ABB RobotStudio station: SJAKKROBOT.rspag

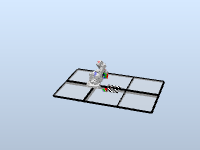
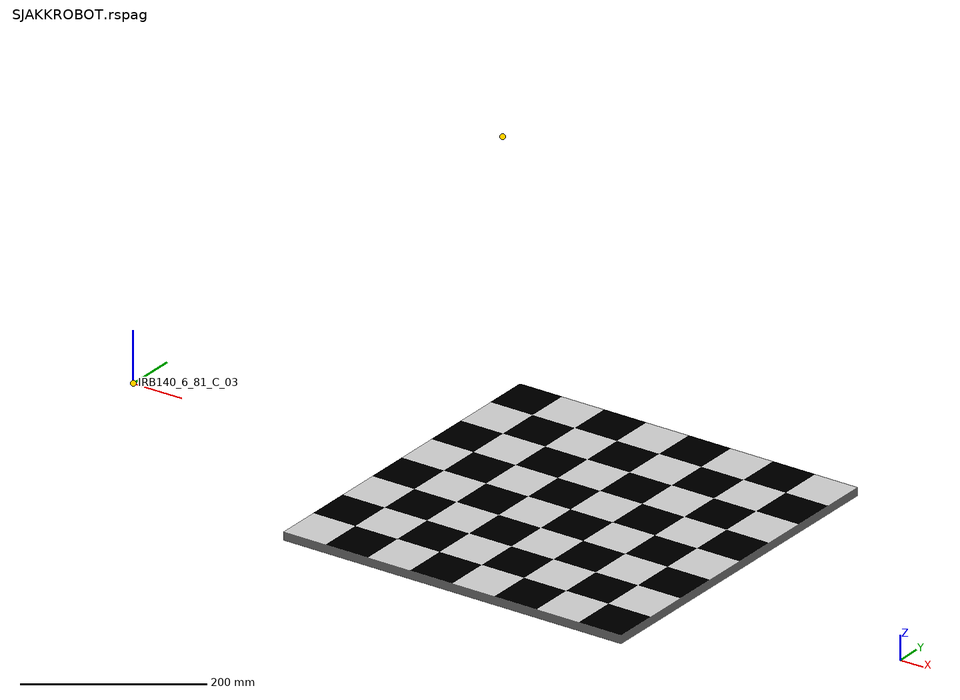
[picture v1: parts stored in the station drawn from their meshes, with robot base, taught points and paths (robot models come from the ABB library and are not in the file)]
--- station ---
Station Solution10 (saved by RobotStudio 21.2.9526.0)
Controller IRB140_6_81
  mechanical unit ROB_1: IRB140_6_81_C_03, 6 joints, base frame (0, 0, 0) mm
Layout (positions relative to the parent item):
  - IRB140_6_81_C_03 [mechanism, from Robots\IRB140_6_81_C_G_03.rslib] at (0, 0, 0) mm; joint values [1.0633, 0.4639, 0.5303, 0, 0.5766, 4.2048] (rad or m)
  - Part_1 [part], size 20 x 20 x 100 mm
  - picker [mechanism] at (210.95, 383, 290.4) mm, rotated rx -180 ry 0 rz 0 deg
      TCP picker at (0, 0, 100) mm
      links: Dummy
  - Brett [part], size 440 x 440 x 9.9 mm
  - 1 [part] at (50, 0, 0) mm, size 55 x 440 x 0 mm
  - 2 [part] at (105, 0, 0) mm, size 55 x 440 x 0 mm
  - 3 [part] at (160, 0, 0) mm, size 55 x 440 x 0 mm
  - 4 [part] at (215, 0, 0) mm, size 55 x 440 x 0 mm
  - 5 [part] at (270, 0, 0) mm, size 55 x 440 x 0 mm
  - 6 [part] at (325, 0, 0) mm, size 55 x 440 x 0 mm
  - 7 [part] at (380, 0, 0) mm, size 55 x 440 x 0 mm
  - 8 [part] at (435, 0, 0) mm, size 55 x 440 x 0 mm
Attachment: picker is attached to IRB140_6_81_C_03 / Link6
Targets, tools, work objects and paths stored in the station and not in the controller backup, written as RAPID:
! task T_ROB1
MODULE Module1
  CONST robtarget Target_10:=[[0,0,0],[1,0,0,0],[0,0,0,0],[9E+09,9E+09,9E+09,9E+09,9E+09,9E+09]];
  CONST robtarget A1:=[[27.5,-412.5,0],[1,0,0,0],[0,0,2,0],[9E+09,9E+09,9E+09,9E+09,9E+09,9E+09]];
  CONST robtarget C1:=[[27.5,-302.5,0],[1,0,0,0],[0,0,2,0],[9E+09,9E+09,9E+09,9E+09,9E+09,9E+09]];
  CONST robtarget D1:=[[27.5,-247.5,0],[1,0,0,0],[0,0,2,0],[9E+09,9E+09,9E+09,9E+09,9E+09,9E+09]];
  CONST robtarget E1:=[[27.5,-192.5,0],[1,0,0,0],[-1,0,1,0],[9E+09,9E+09,9E+09,9E+09,9E+09,9E+09]];
  CONST robtarget F1:=[[27.5,-137.5,0],[1,0,0,0],[-1,0,1,0],[9E+09,9E+09,9E+09,9E+09,9E+09,9E+09]];
  CONST robtarget G1:=[[27.5,-82.5,0],[1,0,0,0],[-1,0,1,0],[9E+09,9E+09,9E+09,9E+09,9E+09,9E+09]];
  CONST robtarget H1:=[[27.5,-27.5,0],[1,0,0,0],[-1,0,1,0],[9E+09,9E+09,9E+09,9E+09,9E+09,9E+09]];
  CONST robtarget A2:=[[82.5,-412.5,0],[1,0,0,0],[0,0,2,0],[9E+09,9E+09,9E+09,9E+09,9E+09,9E+09]];
  CONST robtarget B2:=[[82.5,-357.5,0],[1,0,0,0],[0,0,2,0],[9E+09,9E+09,9E+09,9E+09,9E+09,9E+09]];
  CONST robtarget C2:=[[82.5,-302.5,0],[1,0,0,0],[0,0,2,0],[9E+09,9E+09,9E+09,9E+09,9E+09,9E+09]];
  CONST robtarget D2:=[[82.5,-247.5,0],[1,0,0,0],[0,0,2,0],[9E+09,9E+09,9E+09,9E+09,9E+09,9E+09]];
  CONST robtarget E2:=[[82.5,-192.5,0],[1,0,0,0],[-1,0,1,0],[9E+09,9E+09,9E+09,9E+09,9E+09,9E+09]];
  CONST robtarget F2:=[[82.5,-137.5,0],[1,0,0,0],[-1,0,1,0],[9E+09,9E+09,9E+09,9E+09,9E+09,9E+09]];
  CONST robtarget G2:=[[82.5,-82.5,0],[1,0,0,0],[-1,0,1,0],[9E+09,9E+09,9E+09,9E+09,9E+09,9E+09]];
  CONST robtarget H2:=[[82.5,-27.5,0],[1,0,0,0],[-1,0,1,0],[9E+09,9E+09,9E+09,9E+09,9E+09,9E+09]];
  CONST robtarget A3:=[[137.5,-412.5,0],[1,0,0,0],[0,0,2,0],[9E+09,9E+09,9E+09,9E+09,9E+09,9E+09]];
  CONST robtarget B3:=[[137.5,-357.5,0],[1,0,0,0],[0,0,2,0],[9E+09,9E+09,9E+09,9E+09,9E+09,9E+09]];
  CONST robtarget C3:=[[137.5,-302.5,0],[1,0,0,0],[0,0,2,0],[9E+09,9E+09,9E+09,9E+09,9E+09,9E+09]];
  CONST robtarget D3:=[[137.5,-247.5,0],[1,0,0,0],[0,0,2,0],[9E+09,9E+09,9E+09,9E+09,9E+09,9E+09]];
  CONST robtarget E3:=[[137.5,-192.5,0],[1,0,0,0],[-1,0,1,0],[9E+09,9E+09,9E+09,9E+09,9E+09,9E+09]];
  CONST robtarget F3:=[[137.5,-137.5,0],[1,0,0,0],[-1,0,1,0],[9E+09,9E+09,9E+09,9E+09,9E+09,9E+09]];
  CONST robtarget G3:=[[137.5,-82.5,0],[1,0,0,0],[-1,0,1,0],[9E+09,9E+09,9E+09,9E+09,9E+09,9E+09]];
  CONST robtarget H3:=[[137.5,-27.5,0],[1,0,0,0],[-1,0,1,0],[9E+09,9E+09,9E+09,9E+09,9E+09,9E+09]];
  CONST robtarget A4:=[[192.5,-412.5,0],[1,0,0,0],[0,0,2,0],[9E+09,9E+09,9E+09,9E+09,9E+09,9E+09]];
  CONST robtarget B4:=[[192.5,-357.5,0],[1,0,0,0],[0,0,2,0],[9E+09,9E+09,9E+09,9E+09,9E+09,9E+09]];
  CONST robtarget C4:=[[192.5,-302.5,0],[1,0,0,0],[0,0,2,0],[9E+09,9E+09,9E+09,9E+09,9E+09,9E+09]];
  CONST robtarget D4:=[[192.5,-247.5,0],[1,0,0,0],[0,0,2,0],[9E+09,9E+09,9E+09,9E+09,9E+09,9E+09]];
  CONST robtarget E4:=[[192.5,-192.5,0],[1,0,0,0],[-1,0,1,0],[9E+09,9E+09,9E+09,9E+09,9E+09,9E+09]];
  CONST robtarget F4:=[[192.5,-137.5,0],[1,0,0,0],[-1,0,1,0],[9E+09,9E+09,9E+09,9E+09,9E+09,9E+09]];
  CONST robtarget G4:=[[192.5,-82.5,0],[1,0,0,0],[-1,0,1,0],[9E+09,9E+09,9E+09,9E+09,9E+09,9E+09]];
  CONST robtarget H4:=[[192.5,-27.5,0],[1,0,0,0],[-1,0,1,0],[9E+09,9E+09,9E+09,9E+09,9E+09,9E+09]];
  CONST robtarget A5:=[[247.5,-412.5,0],[1,0,0,0],[0,0,2,0],[9E+09,9E+09,9E+09,9E+09,9E+09,9E+09]];
  CONST robtarget B5:=[[247.5,-357.5,0],[1,0,0,0],[0,0,2,0],[9E+09,9E+09,9E+09,9E+09,9E+09,9E+09]];
  CONST robtarget C5:=[[247.5,-302.5,0],[1,0,0,0],[0,0,2,0],[9E+09,9E+09,9E+09,9E+09,9E+09,9E+09]];
  CONST robtarget D5:=[[247.5,-247.5,0],[1,0,0,0],[0,0,2,0],[9E+09,9E+09,9E+09,9E+09,9E+09,9E+09]];
  CONST robtarget E5:=[[247.5,-192.5,0],[1,0,0,0],[-1,0,1,0],[9E+09,9E+09,9E+09,9E+09,9E+09,9E+09]];
  CONST robtarget F5:=[[247.5,-137.5,0],[1,0,0,0],[-1,0,1,0],[9E+09,9E+09,9E+09,9E+09,9E+09,9E+09]];
  CONST robtarget G5:=[[247.5,-82.5,0],[1,0,0,0],[-1,0,1,0],[9E+09,9E+09,9E+09,9E+09,9E+09,9E+09]];
  CONST robtarget H5:=[[247.5,-27.5,0],[1,0,0,0],[-1,0,1,0],[9E+09,9E+09,9E+09,9E+09,9E+09,9E+09]];
  CONST robtarget A6:=[[302.5,-412.5,0],[1,0,0,0],[0,0,2,0],[9E+09,9E+09,9E+09,9E+09,9E+09,9E+09]];
  CONST robtarget B6:=[[302.5,-357.5,0],[1,0,0,0],[0,0,2,0],[9E+09,9E+09,9E+09,9E+09,9E+09,9E+09]];
  CONST robtarget C6:=[[302.5,-302.5,0],[1,0,0,0],[0,0,2,0],[9E+09,9E+09,9E+09,9E+09,9E+09,9E+09]];
  CONST robtarget D6:=[[302.5,-247.5,0],[1,0,0,0],[0,0,2,0],[9E+09,9E+09,9E+09,9E+09,9E+09,9E+09]];
  CONST robtarget E6:=[[302.5,-192.5,0],[1,0,0,0],[-1,0,1,0],[9E+09,9E+09,9E+09,9E+09,9E+09,9E+09]];
  CONST robtarget F6:=[[302.5,-137.5,0],[1,0,0,0],[-1,0,1,0],[9E+09,9E+09,9E+09,9E+09,9E+09,9E+09]];
  CONST robtarget G6:=[[302.5,-82.5,0],[1,0,0,0],[-1,0,1,0],[9E+09,9E+09,9E+09,9E+09,9E+09,9E+09]];
  CONST robtarget H6:=[[302.5,-27.5,0],[1,0,0,0],[-1,0,1,0],[9E+09,9E+09,9E+09,9E+09,9E+09,9E+09]];
  CONST robtarget A7:=[[357.5,-412.5,0],[1,0,0,0],[0,0,2,0],[9E+09,9E+09,9E+09,9E+09,9E+09,9E+09]];
  CONST robtarget B7:=[[357.5,-357.5,0],[1,0,0,0],[0,0,2,0],[9E+09,9E+09,9E+09,9E+09,9E+09,9E+09]];
  CONST robtarget C7:=[[357.5,-302.5,0],[1,0,0,0],[0,0,2,0],[9E+09,9E+09,9E+09,9E+09,9E+09,9E+09]];
  CONST robtarget D7:=[[357.5,-247.5,0],[1,0,0,0],[0,0,2,0],[9E+09,9E+09,9E+09,9E+09,9E+09,9E+09]];
  CONST robtarget E7:=[[357.5,-192.5,0],[1,0,0,0],[-1,0,1,0],[9E+09,9E+09,9E+09,9E+09,9E+09,9E+09]];
  CONST robtarget F7:=[[357.5,-137.5,0],[1,0,0,0],[-1,0,1,0],[9E+09,9E+09,9E+09,9E+09,9E+09,9E+09]];
  CONST robtarget G7:=[[357.5,-82.5,0],[1,0,0,0],[-1,0,1,0],[9E+09,9E+09,9E+09,9E+09,9E+09,9E+09]];
  CONST robtarget H7:=[[357.5,-27.5,0],[1,0,0,0],[-1,0,1,0],[9E+09,9E+09,9E+09,9E+09,9E+09,9E+09]];
  CONST robtarget A8:=[[412.5,-412.5,0],[1,0,0,0],[0,0,2,0],[9E+09,9E+09,9E+09,9E+09,9E+09,9E+09]];
  CONST robtarget B8:=[[412.5,-357.5,0],[1,0,0,0],[0,0,2,0],[9E+09,9E+09,9E+09,9E+09,9E+09,9E+09]];
  CONST robtarget C8:=[[412.5,-302.5,0],[1,0,0,0],[0,0,2,0],[9E+09,9E+09,9E+09,9E+09,9E+09,9E+09]];
  CONST robtarget D8:=[[412.5,-247.5,0],[1,0,0,0],[0,0,2,0],[9E+09,9E+09,9E+09,9E+09,9E+09,9E+09]];
  CONST robtarget E8:=[[412.5,-192.5,0],[1,0,0,0],[-1,0,1,0],[9E+09,9E+09,9E+09,9E+09,9E+09,9E+09]];
  CONST robtarget F8:=[[412.5,-137.5,0],[1,0,0,0],[-1,0,1,0],[9E+09,9E+09,9E+09,9E+09,9E+09,9E+09]];
  CONST robtarget G8:=[[412.5,-82.5,0],[1,0,0,0],[-1,0,1,0],[9E+09,9E+09,9E+09,9E+09,9E+09,9E+09]];
  CONST robtarget H8:=[[412.5,-27.5,0],[1,0,0,0],[-1,0,1,0],[9E+09,9E+09,9E+09,9E+09,9E+09,9E+09]];
  CONST robtarget B1:=[[27.5,-357.5,0],[1,0,0,0],[0,0,2,0],[9E+09,9E+09,9E+09,9E+09,9E+09,9E+09]];
  VAR robtarget home:=[[192.5,-302.5,-100],[1,0,0,0],[0,0,2,0],[9E+09,9E+09,9E+09,9E+09,9E+09,9E+09]];
  PROC Path_10()
    MoveL A1,v1000,fine,picker\WObj:=board2;
    MoveL A1,v1000,fine,picker\WObj:=board;
    MoveL A1,v1000,fine,picker\WObj:=board2;
    MoveL B1,v1000,fine,picker\WObj:=board2;
    MoveL B1,v1000,fine,picker\WObj:=board;
    MoveL B1,v1000,fine,picker\WObj:=board2;
    MoveL C1,v1000,fine,picker\WObj:=board2;
    MoveL C1,v1000,fine,picker\WObj:=board;
    MoveL C1,v1000,fine,picker\WObj:=board2;
    MoveL D1,v1000,fine,picker\WObj:=board2;
    MoveL D1,v1000,fine,picker\WObj:=board;
    MoveL D1,v1000,fine,picker\WObj:=board2;
    MoveL E1,v1000,fine,picker\WObj:=board2;
    MoveL E1,v1000,fine,picker\WObj:=board;
    MoveL E1,v1000,fine,picker\WObj:=board2;
    MoveL F1,v1000,fine,picker\WObj:=board2;
    MoveL F1,v1000,fine,picker\WObj:=board;
    MoveL F1,v1000,fine,picker\WObj:=board2;
    MoveL G1,v1000,fine,picker\WObj:=board2;
    MoveL G1,v1000,fine,picker\WObj:=board;
    MoveL G1,v1000,fine,picker\WObj:=board2;
    MoveL H1,v1000,fine,picker\WObj:=board2;
    MoveL H1,v1000,fine,picker\WObj:=board;
    MoveL H1,v1000,fine,picker\WObj:=board2;
    MoveL A2,v1000,fine,picker\WObj:=board2;
    MoveL A2,v1000,fine,picker\WObj:=board;
    MoveL A2,v1000,fine,picker\WObj:=board2;
    MoveL B2,v1000,fine,picker\WObj:=board2;
    MoveL B2,v1000,fine,picker\WObj:=board;
    MoveL B2,v1000,fine,picker\WObj:=board2;
    MoveL C2,v1000,fine,picker\WObj:=board2;
    MoveL C2,v1000,fine,picker\WObj:=board;
    MoveL C2,v1000,fine,picker\WObj:=board2;
    MoveL D2,v1000,fine,picker\WObj:=board2;
    MoveL D2,v1000,fine,picker\WObj:=board;
    MoveL D2,v1000,fine,picker\WObj:=board2;
    MoveL E2,v1000,fine,picker\WObj:=board2;
    MoveL E2,v1000,fine,picker\WObj:=board;
    MoveL E2,v1000,fine,picker\WObj:=board2;
    MoveL F2,v1000,fine,picker\WObj:=board2;
    MoveL F2,v1000,fine,picker\WObj:=board;
    MoveL F2,v1000,fine,picker\WObj:=board2;
    MoveL G2,v1000,fine,picker\WObj:=board2;
    MoveL G2,v1000,fine,picker\WObj:=board;
    MoveL G2,v1000,fine,picker\WObj:=board2;
    MoveL H2,v1000,fine,picker\WObj:=board2;
    MoveL H2,v1000,fine,picker\WObj:=board;
    MoveL H2,v1000,fine,picker\WObj:=board2;
    MoveL A3,v1000,fine,picker\WObj:=board2;
    MoveL A3,v1000,fine,picker\WObj:=board;
    MoveL A3,v1000,fine,picker\WObj:=board2;
    MoveL B3,v1000,fine,picker\WObj:=board2;
    MoveL B3,v1000,fine,picker\WObj:=board;
    MoveL B3,v1000,fine,picker\WObj:=board2;
    MoveL C3,v1000,fine,picker\WObj:=board2;
    MoveL C3,v1000,fine,picker\WObj:=board;
    MoveL C3,v1000,fine,picker\WObj:=board2;
    MoveL D3,v1000,fine,picker\WObj:=board2;
    MoveL D3,v1000,fine,picker\WObj:=board;
    MoveL D3,v1000,fine,picker\WObj:=board2;
    MoveL E3,v1000,fine,picker\WObj:=board2;
    MoveL E3,v1000,fine,picker\WObj:=board;
    MoveL E3,v1000,fine,picker\WObj:=board2;
    MoveL F3,v1000,fine,picker\WObj:=board2;
    MoveL F3,v1000,fine,picker\WObj:=board;
    MoveL F3,v1000,fine,picker\WObj:=board2;
    MoveL G3,v1000,fine,picker\WObj:=board2;
    MoveL G3,v1000,fine,picker\WObj:=board;
    MoveL G3,v1000,fine,picker\WObj:=board2;
    MoveL H3,v1000,fine,picker\WObj:=board2;
    MoveL H3,v1000,fine,picker\WObj:=board;
    MoveL H3,v1000,fine,picker\WObj:=board2;
    MoveL A4,v1000,fine,picker\WObj:=board2;
    MoveL A4,v1000,fine,picker\WObj:=board;
    MoveL A4,v1000,fine,picker\WObj:=board2;
    MoveL B4,v1000,fine,picker\WObj:=board2;
    MoveL B4,v1000,fine,picker\WObj:=board;
    MoveL B4,v1000,fine,picker\WObj:=board2;
    MoveL C4,v1000,fine,picker\WObj:=board2;
    MoveL C4,v1000,fine,picker\WObj:=board;
    MoveL C4,v1000,fine,picker\WObj:=board2;
    MoveL D4,v1000,fine,picker\WObj:=board2;
    MoveL D4,v1000,fine,picker\WObj:=board;
    MoveL D4,v1000,fine,picker\WObj:=board2;
    MoveL E4,v1000,fine,picker\WObj:=board2;
    MoveL E4,v1000,fine,picker\WObj:=board;
    MoveL E4,v1000,fine,picker\WObj:=board2;
    MoveL F4,v1000,fine,picker\WObj:=board2;
    MoveL F4,v1000,fine,picker\WObj:=board;
    MoveL F4,v1000,fine,picker\WObj:=board2;
    MoveL G4,v1000,fine,picker\WObj:=board2;
    MoveL G4,v1000,fine,picker\WObj:=board;
    MoveL G4,v1000,fine,picker\WObj:=board2;
    MoveL H4,v1000,fine,picker\WObj:=board2;
    MoveL H4,v1000,fine,picker\WObj:=board;
    MoveL H4,v1000,fine,picker\WObj:=board2;
    MoveL A5,v1000,fine,picker\WObj:=board2;
    MoveL A5,v1000,fine,picker\WObj:=board;
    MoveL A5,v1000,fine,picker\WObj:=board2;
    MoveL B5,v1000,fine,picker\WObj:=board2;
    MoveL B5,v1000,fine,picker\WObj:=board;
    MoveL B5,v1000,fine,picker\WObj:=board2;
    MoveL C5,v1000,fine,picker\WObj:=board2;
    MoveL C5,v1000,fine,picker\WObj:=board;
    MoveL C5,v1000,fine,picker\WObj:=board2;
    MoveL D5,v1000,fine,picker\WObj:=board2;
    MoveL D5,v1000,fine,picker\WObj:=board;
    MoveL D5,v1000,fine,picker\WObj:=board2;
    MoveL E5,v1000,fine,picker\WObj:=board2;
    MoveL E5,v1000,fine,picker\WObj:=board;
    MoveL E5,v1000,fine,picker\WObj:=board2;
    MoveL F5,v1000,fine,picker\WObj:=board2;
    MoveL F5,v1000,fine,picker\WObj:=board;
    MoveL F5,v1000,fine,picker\WObj:=board2;
    MoveL G5,v1000,fine,picker\WObj:=board2;
    MoveL G5,v1000,fine,picker\WObj:=board;
    MoveL G5,v1000,fine,picker\WObj:=board2;
    MoveL H5,v1000,fine,picker\WObj:=board2;
    MoveL H5,v1000,fine,picker\WObj:=board;
    MoveL H5,v1000,fine,picker\WObj:=board2;
    MoveL A6,v1000,fine,picker\WObj:=board2;
    MoveL A6,v1000,fine,picker\WObj:=board;
    MoveL A6,v1000,fine,picker\WObj:=board2;
    MoveL B6,v1000,fine,picker\WObj:=board2;
    MoveL B6,v1000,fine,picker\WObj:=board;
    MoveL B6,v1000,fine,picker\WObj:=board2;
    MoveL C6,v1000,fine,picker\WObj:=board2;
    MoveL C6,v1000,fine,picker\WObj:=board;
    MoveL C6,v1000,fine,picker\WObj:=board2;
    MoveL D6,v1000,fine,picker\WObj:=board2;
    MoveL D6,v1000,fine,picker\WObj:=board;
    MoveL D6,v1000,fine,picker\WObj:=board2;
    MoveL E6,v1000,fine,picker\WObj:=board2;
    MoveL E6,v1000,fine,picker\WObj:=board;
    MoveL E6,v1000,fine,picker\WObj:=board2;
    MoveL F6,v1000,fine,picker\WObj:=board2;
    MoveL F6,v1000,fine,picker\WObj:=board;
    MoveL F6,v1000,fine,picker\WObj:=board2;
    MoveL G6,v1000,fine,picker\WObj:=board2;
    MoveL G6,v1000,fine,picker\WObj:=board;
    MoveL G6,v1000,fine,picker\WObj:=board2;
    MoveL H6,v1000,fine,picker\WObj:=board2;
    MoveL H6,v1000,fine,picker\WObj:=board;
    MoveL H6,v1000,fine,picker\WObj:=board2;
    MoveL A7,v1000,fine,picker\WObj:=board2;
    MoveL A7,v1000,fine,picker\WObj:=board;
    MoveL A7,v1000,fine,picker\WObj:=board2;
    MoveL B7,v1000,fine,picker\WObj:=board2;
    MoveL B7,v1000,fine,picker\WObj:=board;
    MoveL B7,v1000,fine,picker\WObj:=board2;
    MoveL C7,v1000,fine,picker\WObj:=board2;
    MoveL C7,v1000,fine,picker\WObj:=board;
    MoveL C7,v1000,fine,picker\WObj:=board2;
    MoveL D7,v1000,fine,picker\WObj:=board2;
    MoveL D7,v1000,fine,picker\WObj:=board;
    MoveL D7,v1000,fine,picker\WObj:=board2;
    MoveL E7,v1000,fine,picker\WObj:=board2;
    MoveL E7,v1000,fine,picker\WObj:=board;
    MoveL E7,v1000,fine,picker\WObj:=board2;
    MoveL F7,v1000,fine,picker\WObj:=board2;
    MoveL F7,v1000,fine,picker\WObj:=board;
    MoveL F7,v1000,fine,picker\WObj:=board2;
    MoveL G7,v1000,fine,picker\WObj:=board2;
    MoveL G7,v1000,fine,picker\WObj:=board;
    MoveL G7,v1000,fine,picker\WObj:=board2;
    MoveL H7,v1000,fine,picker\WObj:=board2;
    MoveL H7,v1000,fine,picker\WObj:=board;
    MoveL H7,v1000,fine,picker\WObj:=board2;
    MoveL A8,v1000,fine,picker\WObj:=board2;
    MoveL A8,v1000,fine,picker\WObj:=board;
    MoveL A8,v1000,fine,picker\WObj:=board2;
    MoveL B8,v1000,fine,picker\WObj:=board2;
    MoveL B8,v1000,fine,picker\WObj:=board;
    MoveL B8,v1000,fine,picker\WObj:=board2;
    MoveL C8,v1000,fine,picker\WObj:=board2;
    MoveL C8,v1000,fine,picker\WObj:=board;
    MoveL C8,v1000,fine,picker\WObj:=board2;
    MoveL D8,v1000,fine,picker\WObj:=board2;
    MoveL D8,v1000,fine,picker\WObj:=board;
    MoveL D8,v1000,fine,picker\WObj:=board2;
    MoveL E8,v1000,fine,picker\WObj:=board2;
    MoveL E8,v1000,fine,picker\WObj:=board;
    MoveL E8,v1000,fine,picker\WObj:=board2;
    MoveL F8,v1000,fine,picker\WObj:=board2;
    MoveL F8,v1000,fine,picker\WObj:=board;
    MoveL F8,v1000,fine,picker\WObj:=board2;
    MoveL G8,v1000,fine,picker\WObj:=board2;
    MoveL G8,v1000,fine,picker\WObj:=board;
    MoveL G8,v1000,fine,picker\WObj:=board2;
    MoveL H8,v1000,fine,picker\WObj:=board2;
    MoveL H8,v1000,fine,picker\WObj:=board;
    MoveL H8,v1000,fine,picker\WObj:=board2;
  ENDPROC
ENDMODULE

! task T_ROB1
MODULE Tillegg
  PROC Flytt()
    Move;
  ENDPROC
ENDMODULE


--- Backups/IRB140_6_81/RAPID/TASK1/PROGMOD/Brikker_felter.mod ---
MODULE Brikker_felter

        ! Denne prosessen brukes til å gi alle brikken sin utgangsposisjon og høyde, da høyden er ulik for bønner og offiserer.
    PROC brikker()
         brikke{1}:=Offs(TargetA{1}.target,0,0,-Hoyde_OF_S);
         brikke{2}:=Offs(TargetA{2}.target,0,0,-Hoyde_OF_S);
         brikke{3}:=Offs(TargetA{3}.target,0,0,-Hoyde_OF_S);
         brikke{4}:=Offs(TargetA{4}.target,0,0,-Hoyde_OF_S);
         brikke{5}:=Offs(TargetA{5}.target,0,0,-Hoyde_OF_S);
         brikke{6}:=Offs(TargetA{6}.target,0,0,-Hoyde_OF_S);
         brikke{7}:=Offs(TargetA{7}.target,0,0,-Hoyde_OF_S);
         brikke{8}:=Offs(TargetA{8}.target,0,0,-Hoyde_OF_S);
         brikke{9}:=Offs(TargetA{9}.target,0,0,-Hoyde_BO_S);
         brikke{10}:=Offs(TargetA{10}.target,0,0,-Hoyde_BO_S);
         brikke{11}:=Offs(TargetA{11}.target,0,0,-Hoyde_BO_S);
         brikke{12}:=Offs(TargetA{12}.target,0,0,-Hoyde_BO_S);
         brikke{13}:=Offs(TargetA{13}.target,0,0,-Hoyde_BO_S);
         brikke{14}:=Offs(TargetA{14}.target,0,0,-Hoyde_BO_S);
         brikke{15}:=Offs(TargetA{15}.target,0,0,-Hoyde_BO_S);
         brikke{16}:=Offs(TargetA{16}.target,0,0,-Hoyde_BO_S);

         brikke{17}:=Offs(TargetA{49}.target,0,0,-Hoyde_BO_H);
         brikke{18}:=Offs(TargetA{50}.target,0,0,-Hoyde_BO_H);
         brikke{19}:=Offs(TargetA{51}.target,0,0,-Hoyde_BO_H);
         brikke{20}:=Offs(TargetA{52}.target,0,0,-Hoyde_BO_H);
         brikke{21}:=Offs(TargetA{53}.target,0,0,-Hoyde_BO_H);
         brikke{22}:=Offs(TargetA{54}.target,0,0,-Hoyde_BO_H);
         brikke{23}:=Offs(TargetA{55}.target,0,0,-Hoyde_BO_H);
         brikke{24}:=Offs(TargetA{56}.target,0,0,-Hoyde_BO_H);
         brikke{25}:=Offs(TargetA{57}.target,0,0,-Hoyde_OF_H);
         brikke{26}:=Offs(TargetA{58}.target,0,0,-Hoyde_OF_H);
         brikke{27}:=Offs(TargetA{59}.target,0,0,-Hoyde_OF_H);
         brikke{28}:=Offs(TargetA{60}.target,0,0,-Hoyde_OF_H);
         brikke{29}:=Offs(TargetA{61}.target,0,0,-Hoyde_OF_H);
         brikke{30}:=Offs(TargetA{62}.target,0,0,-Hoyde_OF_H);
         brikke{31}:=Offs(TargetA{63}.target,0,0,-Hoyde_OF_H);
         brikke{32}:=Offs(TargetA{64}.target,0,0,-Hoyde_OF_H);

         ENDPROC


    ! Denne prosessen setter kordinatene til alle feltene
    PROC Felt()
        CONST num felt := 434/8; !bredden per felt

        ! Felt 1, er i i 0,0,0 ut i fra Workobjectet
        TargetA{1}.target:=[[0,0,0],[1,0,0,0],[0,0,2,0],[9E+9,9E+9,9E+9,9E+9,9E+9,9E+9]];

        ! Setter rader og kolonner med disse to for-løkkene
        FOR i FROM 1 TO 8 DO
            FOR j FROM 1 TO 8 DO
                TargetA{j+(i-1)*8}.target:=Offs(TargetA{1}.target,(i-1)*felt,-(j-1)*felt,0);
            ENDFOR
        ENDFOR
    ENDPROC

ENDMODULE

--- Backups/IRB140_6_81/RAPID/TASK1/PROGMOD/CalibData.mod ---
MODULE CalibData
    PERS tooldata picker:=[TRUE,[[0,0,90.4],[1,0,0,0]],[1,[0,0,1],[1,0,0,0],0,0,0]];
    TASK PERS wobjdata board:=[FALSE,TRUE,"",[[363.9,-176.7,20],[0,1,0,0]],[[0,0,0],[1,0,0,0]]];
    TASK PERS wobjdata board2:=[FALSE,TRUE,"",[[363.9,-176.7,20],[0,1,0,0]],[[0,0,0],[1,0,0,0]]];
    TASK PERS wobjdata safepose:=[FALSE,TRUE,"",[[213,383,200],[0,1,0,0]],[[0,0,0],[1,0,0,0]]];
ENDMODULE

--- Backups/IRB140_6_81/RAPID/TASK1/PROGMOD/Ikke_i_bruk.mod ---
MODULE Ikke_i_bruk

    PROC Oppsett ()
    VAR num knapp:=0;
    WHILE knapp <5 DO
        TPReadFK knapp, "Trykk","A8","H8","A1","H1","Start spill";
        IF knapp=1 THEN
            MoveJ Offs(TargetA{1}.target,0,0,-35),Speed_hor,fine,picker\WObj:=board2;
        ELSEIF knapp=2 THEN
            MoveJ Offs(TargetA{8}.target,0,0,-35),Speed_hor,fine,picker\WObj:=board2;
        ELSEIF knapp=3 THEN
            MoveJ Offs(TargetA{57}.target,0,0,-35),Speed_hor,fine,picker\WObj:=board2;
        ELSEIF knapp=4 THEN
            MoveJ Offs(TargetA{64}.target,0,0,-35),Speed_hor,fine,picker\WObj:=board2;
        ELSEIF knapp=5 THEN
            safe_pose;
        ENDIF
    ENDWHILE
    ENDPROC

     PROC aaa_test()
    !mm:= 1;
    !P1_x:=0;
    !P1_y:=0;
    data:="sc,0,4,0,2";
    sjekk_string;
    !data:="b3333,385,220;385,110";

    data:="b3333,220,385;110,385";
    sjekk_string;
    WaitTime(2);
    data:="rc";
    sjekk_string;
    data:="b3333,110,385;220,385";
    sjekk_string;
    WaitTime(2);
    data:="rc";
    sjekk_string;
    data:="b3333,220,385;330,385";
    sjekk_string;
    WaitTime(2);
    data:="rc";
    sjekk_string;




    WaitTime(5);
    ENDPROC

    ! Denne prosedyren setter brikker tilbake på sin egenplass.
    PROC clean()
        VAR num k:=0;
        VAR num p:=17;
        VAR num th:=5;

        ! Flytter brikke fra 1 til 32 tilbake på plass
        FOR i FROM 1 TO 32 DO
            Opptatt;
            ! hvis i er over 16 blir k:=i+32, dette er for at å plasere brikken på riktig rute
            IF i>16 THEN
                k:=i+32;
            ELSE
                k:=i;
            ENDIF

            ! hvis brikke står innenfor th,mm fra sin riktige plass skal den ikke flyttets på.
                IF NOT (TargetA{k}.target.trans.x-th < brikke{i}.trans.x  AND  TargetA{k}.target.trans.x + th > brikke{i}.trans.x AND TargetA{k}.target.trans.y-th < brikke{i}.trans.y  AND  TargetA{k}.target.trans.y + th > brikke{i}.trans.y) THEN

                    ! Hvis plassen brikke skal til er opptatt må den til en "lagerplass" får den kan plaseres riktig
                    IF  TargetA{k}.opptatt THEN
                        ! Sjekker om "lagerplassen" er opptatt frem til den finner en plass som er ledig
                        WHILE NOT TargetA{p}.opptatt DO
                            IF TargetA{p}.opptatt THEN
                                p:=p+1;
                            ENDIF
                        ENDWHILE

                        ! Gir riktig verdi til de globale variable og flytter brikken
                        brikke_flytt:=i;
                        Til_felt:=p;
                        Move;

                    ! Hvis plassen er ledig gjøres denne prosessen, gir riktig verdi til de globale variable og flytter brikken
                    ELSEIF NOT TargetA{k}.opptatt THEN
                        brikke_flytt:=i;
                        Til_felt:=k;
                        Move;
                ENDIF
            ENDIF
        ENDFOR
    ENDPROC

        ! Denne prosessen mottar hvor mange mm en pixel er og posisjonen til en kjent brikke.
    PROC Motta_mm_pos()
        VAR string mm_s:="";
        VAR string p1x_s:="";
        VAR string p1y_s:="";
        VAR bool ok;
        VAR string id3;
        id3:=data;

        ! Deler opp stringen i de ulike delene,
        ! Dette er bestemt på forhånd hvordan denne skal se ut
        mm_s := StrPart(id3,1,6);
        p1x_s := StrPart(id3,8,4);
        p1y_s := StrPart(id3,13,4);

        ! Fra string til NUM
        ok := StrToVal(mm_s,mm);
        ok := StrToVal(p1x_s,P1_x);
        ok := StrToVal(p1y_s,P1_y);
    ENDPROC

    PROC Motta_id()
        VAR string id_s:="";
        VAR string x_s:="";
        VAR string y_s:="";
        VAR num id_n:=0;
        VAR num x_n:=0;
        VAR num y_n:=0;
        VAR bool ok;
        VAR string id1;
        id1:=data;

        FOR i FROM 1 TO 2 DO

        ! Deler opp i Brikke ID, X og Y verdi i pixel
        id_s := StrPart(id1,1+(i-1)*13,2);  ! Finner brikke ID
        x_s := StrPart(id1,4+(i-1)*13,4);   ! Finner X i pixel
        y_s := StrPart(id1,9+(i-1)*13,4);   ! Finner Y i pixel


        TPWrite id_s + " " + x_s + " " + y_s;   ! Skriver ut til flexpedant
        ok := StrToVal(id_s,id_n);              ! ID til NUM
        ok := StrToVal(x_s,x_n);                ! X til NUM
        ok := StrToVal(y_s,y_n);                ! Y til NUM

        ! Lagrer posisjonen til brikken i riktig brikke med brikke-ID og gjør matten for hvor brikken er
        ! (x_n-P1_x)*mm: x_n er pixelverdi til denne brikken, P1_x er pixelverdi til brikken som står i 0,0,0mi forhold til workobjektet. mm er milimeter verdi
        brikke{id_n}:=[[(x_n-P1_x)*mm,(y_n-P1_y)*mm,brikke{id_n}.trans.z],[1,0,0,0],[0,0,2,0],[9E+9,9E+9,9E+9,9E+9,9E+9,9E+9]];

        ENDFOR
    ENDPROC


ENDMODULE

--- Backups/IRB140_6_81/RAPID/TASK1/PROGMOD/Module1.mod ---
MODULE Module1
    RECORD cell
        robtarget target;
        bool opptatt;
    ENDRECORD

    const speeddata Speed_opp := v100;
    const speeddata Speed_ned := v50;
    const speeddata Speed_hor := v200;
    const num tid:=0.5;

    VAR cell TargetA{64};
    VAR robtarget brikke{34};

    VAR num mm:= 0.5841;
    VAR num P1_x:=127;
    VAR num P1_y:=131;
    VAR num frax:= 0;
    VAR num fray:=0;
    VAR num tilx:=0;
    VAR num tily:=0;

    ! Høyde til brikkene
    CONST NUM Hoyde_OF_H := 30; ! Hvit offiser
    CONST NUM Hoyde_BO_H := 20; ! Hvit bonde
    CONST NUM Hoyde_OF_S := 26; ! Svart offiser
    CONST NUM Hoyde_BO_S := 20; ! Svart bonde

    VAR intnum Hold1;
    VAR intnum Hold2;
    VAR NUM HOLD:=0;

    !*******************************
    VAR socketdev server;
    VAR socketdev client;
    VAR string Client_IP;
    VAR string data := "";
    VAR string msg := "Client hello"; ! Dette er stringen som brukes til å sende tilbake til Python


    !Vars for hjelpefunksjon
    VAR num j;
    VAR num i;
    VAR num x;
    VAR num k;
    VAR num brikke_ut:= 0;
    VAR num f;  !fra
    VAR num t;  !til
    var num brikke_flytt;
    var num Til_felt;
    var num fra_felt;
    VAR num lager1:=0;
    VAR num lager2:=1;

    PROC main()
        ConfL \Off;
        ConfJ \Off;
        safe_pose;
        Felt;
        brikker;

        ! Dette er for interrupt rutine
        CONNECT Hold1 WITH rutine1;
        ISignalDI DI10_1 ,1,Hold1;
        CONNECT Hold2 WITH rutine2;
        ISignalDI DI10_2 ,1,Hold2;

        ! Oppsett av server instilliger
        SocketCreate server;
        SocketBind server, "192.168.12.57",2222;
        SocketListen server;
        SocketAccept server, client, \ClientAddress:=Client_IP\Time:=120;

        !Svarer klienten
        TPWrite "Client_IP: " + Client_IP;
        msg := "Client hello";
        SocketSend client \Str:=msg;

        !Main Loop
        WHILE data <> "EXIT" DO
            !Venter på komando
            SocketReceive client \Str:=data;
            TPWrite "Data motatt: " + data;
            sjekk_string;
        ENDWHILE

        SocketClose server;
        SocketClose client;

    ENDPROC

! Disse TRAP funksjonen brukes for å få roboten ut av WHILE-loopen som gjør det trygt å flytte en brikke
TRAP rutine1
   HOLD:=1;
ENDTRAP

TRAP rutine2
    HOLD:=1;
ENDTRAP

ENDMODULE

--- Backups/IRB140_6_81/RAPID/TASK1/PROGMOD/String_behandling.mod ---
MODULE String_behandling

    PROC sjekk_string()
            ! Mottar at trekket er riktig og lagrer posisjonen til den hvite brikke som er flytet.
        IF "r" = StrPart(data,1,1) THEN
            msg:="r";
            lagre_hvit_flytt;
            TPWrite msg;
            SocketSend client \Str:=msg;

            ! Mottar posisjon til hvit trekk og sender tilbake feltet som brikken har flytett seg til.
        ELSEIF "b" = StrPart(data,1,1) THEN
            motta_hvit_flytt;
            SocketSend client \Str:=msg;
            TPWrite msg;


            ! Flytter roboten til safe_pose og setter roboten til en "hold" loop,
            ! som kun kan gå ut av ved å trykke på knappen ved siden eller
        ELSEIF "k" = StrPart(data,1,1) THEN
            safe_pose;
            while_hold;
            msg:="OKBilde";
            TPWrite msg;
            SocketSend client \Str:=msg;

            ! Trekket som ble gjort var ulovlig og skriver ut på FlexPedanten.
        ELSEIF "f" = StrPart(data,1,1) THEN
            TPWrite "Ulovlig trekk, flytt brikken(e) tilbake.";

            ! Svart i trekk her er det også lagt
        ELSEIF "s" = StrPart(data,1,1) THEN
            IF "r" = StrPart(data,2,1) THEN
                motta_svart_move;

                ! Sjekker om det er Rokade
            ELSEIF "c" = StrPart(data,2,1) THEN
                motta_svart_move;
                ! Sjekker hvilken vei kongen gikk
                IF brikke_flytt<Til_felt THEN
                    brikke_flytt:=8;
                    Til_felt:=6;
                ELSE
                    brikke_flytt:=1;
                    Til_felt:=4;
                ENDIF
                spille;

                ! Sjekker om det er en passant
            ELSEIF "e" = StrPart(data,2,1) THEN
                ! Siden det er kun lov med dette trekke rett etter at en bonde har gått 2 frem vil denne brikke forsatt være lagret her.
                brikke_ut:=brikke_flytt;
                Sla_ut;
                motta_svart_move;
            ENDIF

                safe_pose;
                msg:="OKBilde";
            TPWrite msg;
            SocketSend client \Str:=msg;
        ENDIF
    ENDPROC

    ! Denne er for lagre verdien til den hvite brikke som akkurat ble flyttet hvis trekke var lovlig.
    PROC lagre_hvit_flytt()
        VAR num th:=20;



         FOR i FROM 17 TO 32 DO
            ! Finner brikken.
                IF TargetA{fra_felt}.target.trans.x-th < brikke{i}.trans.x  AND  TargetA{fra_felt}.target.trans.x + th > brikke{i}.trans.x AND TargetA{fra_felt}.target.trans.y-th < brikke{i}.trans.y  AND  TargetA{fra_felt}.target.trans.y + th > brikke{i}.trans.y THEN

                        ! hvis kongen som er brikke 29 flytter seg mer en 1 plass i y rettning lagres tårnet til riktig plass.
                            IF i=29 and brikke{29}.trans.y > brikke{33}.trans.y + 80  and "c" = StrPart(data,2,1) THEN
                                brikke{32}:= TargetA{62}.target;
                                TPWrite "Kort rokade";
                            ELSEIF i=29 and brikke{29}.trans.y < brikke{33}.trans.y - 80 and "c" = StrPart(data,2,1) THEN
                                brikke{25}:= TargetA{59}.target;
                                TPWrite "Lang rokade";
                            ENDIF

                        brikke{i}:= Offs(brikke{33},0,0,brikke{i}.trans.z);
                ENDIF
         ENDFOR

        ! Hvis svart brikke blir slått ut blir posisjonen satt på utsiden av brettet slik at den ikke kan forstyrre spillet.
            FOR i FROM 1 TO 16 DO
            ! Finner brikken.
                IF brikke{33}.trans.x-th < brikke{i}.trans.x  AND  brikke{33}.trans.x + th > brikke{i}.trans.x AND brikke{33}.trans.y-th < brikke{i}.trans.y  AND  brikke{33}.trans.y + th > brikke{i}.trans.y THEN
                        brikke{i}:=OFFS(TargetA{8}.target,-100,-100,brikke{i}.trans.z);
                ENDIF
        ENDFOR

        ! Sjekker om det er en passant
        IF "e" = StrPart(data,2,1) THEN
            FOR i FROM 1 TO 16 DO
                IF brikke{34}= brikke{i} THEN
                    brikke{i}:=OFFS(TargetA{8}.target,-100,-100,brikke{i}.trans.z);
                ENDIF
            ENDFOR
        ENDIF

        Opptatt;
    ENDPROC

    PROC motta_svart_move()
        VAR string x_s:="";
        VAR string y_s:="";
        VAR string z_s:="";
        VAR string p_s:="";
        VAR num x_n;
        VAR num y_n;
        VAR num z_n;
        VAR num p_n;
        VAR bool ok;
        VAR num fra_felt;
        VAR num th:=20;


        x_s := StrPart(data,4,1);
        y_s := StrPart(data,6,1);
        z_s := StrPart(data,8,1);
        p_s := StrPart(data,10,1);

        ok := StrToVal(x_s,x_n);
        ok := StrToVal(y_s,y_n);
        ok := StrToVal(z_s,z_n);
        ok := StrToVal(p_s,p_n);

        fra_felt:= x_n*8+(y_n+1);
        Til_felt:= z_n*8+(p_n+1);

            FOR i FROM 1 TO 32 DO
                IF (TargetA{fra_felt}.target.trans.x-th < brikke{i}.trans.x  AND  TargetA{fra_felt}.target.trans.x + th > brikke{i}.trans.x AND TargetA{fra_felt}.target.trans.y-th < brikke{i}.trans.y  AND  TargetA{fra_felt}.target.trans.y + th > brikke{i}.trans.y) THEN
                    brikke_flytt:=i;
                ENDIF
            ENDFOR
        ! Kjører spill
        spille;
    ENDPROC

    !Denne prosessen mottar string fra python og brukes til å flytte brikker fra et punkt til et annet.
    PROC motta_hvit_flytt ()
        VAR string frax_s:="";
        VAR string fray_s:="";
        VAR string tilx_s:="";
        VAR string tily_s:="";
        VAR bool ok;
        VAR num length_n{4};
        VAR num th:=20;
        VAR string length_s{4};
        VAR string til_s;
        VAR string fra_s;
        VAR num til_n:=0;
        VAR num fra_n:=0;
        VAR string id2;   ! flytting
        id2:=data;


        FOR i FROM 1 TO 4 DO
            length_s{i} := StrPart(data,1+i,1);
            ok := StrToVal(length_s{i},length_n{i});
        ENDFOR

        ! Deler opp stringen i de ulike kordinatene,
        ! Dette er bestemt på forhånd hvordan denne skal se ut
        frax_s := StrPart(data,7,length_n{1});
        fray_s := StrPart(data,7+1+length_n{1},length_n{2});
        tilx_s := StrPart(data,7+2+length_n{1}+length_n{2},length_n{3});
        tily_s := StrPart(data,7+3+length_n{1}+length_n{2}+length_n{3},length_n{4});

        ! Fra string til NUM
        ok := StrToVal(frax_s,frax);
        ok := StrToVal(fray_s,fray);
        ok := StrToVal(tilx_s,tilx);
        ok := StrToVal(tily_s,tily);
        TPWrite tilx_s+" " \Num:=tilx;
        FOR i FROM 1 TO 64 DO
            IF (frax-P1_x)*mm-th < -TargetA{i}.target.trans.y  AND  (frax-P1_x)*mm + th > -TargetA{i}.target.trans.y AND (fray-P1_y)*mm-th < TargetA{i}.target.trans.x  AND  (fray-P1_y)*mm + th > TargetA{i}.target.trans.x THEN
                fra_n:=i;
                fra_felt:=i;
            ENDIF
            IF (tilx-P1_x)*mm-th < -TargetA{i}.target.trans.y  AND  (tilx-P1_x)*mm + th > -TargetA{i}.target.trans.y AND (tily-P1_y)*mm-th < TargetA{i}.target.trans.x  AND  (tily-P1_y)*mm + th > TargetA{i}.target.trans.x THEN
                til_n:=i;
            ENDIF
        ENDFOR

fra_s := NumToStr(fra_n,0);
til_s := NumToStr(til_n,0);
msg := fra_s+";"+ til_s;

    brikke{33}:= Offs(TargetA{1}.target,(tily-P1_y)*mm,-(tilx-P1_x)*mm,0);

    ENDPROC

ENDMODULE

--- Backups/IRB140_6_81/RAPID/TASK1/PROGMOD/Tillegg.mod ---
MODULE Tillegg

! Dette er prossen som flytter brikker fra A til B
    PROC Move()


        ! Henter brikke som skal flyttes
        MoveJ Offs(brikke{brikke_flytt},0,0,-100-brikke{brikke_flytt}.trans.z),Speed_hor,fine,picker\WObj:=board2;
        MoveL brikke{brikke_flytt},Speed_ned,fine,picker\WObj:=board2;
        Set DO10_1;
        WaitTime(tid);

        !Flytter brikke til gitt plass
        MoveL Offs(brikke{brikke_flytt},0,0,-100-brikke{brikke_flytt}.trans.z),Speed_opp,fine,picker\WObj:=board2;
        MoveL Offs(TargetA{Til_felt}.target,0,0,-100),Speed_hor,fine,picker\WObj:=board2;
        MoveL Offs(TargetA{Til_felt}.target,0,0,brikke{brikke_flytt}.trans.z),Speed_ned,fine,picker\WObj:=board2;
        reset DO10_1;
        WaitTime(tid);
        MoveL Offs(TargetA{Til_felt}.target,0,0,-100),Speed_opp,fine,picker\WObj:=board2;

        ! Lagrer brikkens nye posisjon
        brikke{brikke_flytt}:=OFFS(TargetA{Til_felt}.target,0,0,brikke{brikke_flytt}.trans.z);
        brikke{34}:=brikke{brikke_flytt}; ! Lagree forrige svart brikke
        ! Setter at fletet er opptatt
        TargetA{Til_felt}.opptatt:=TRUE;

        TPWrite "brikke_flytt=" \Num:=brikke_flytt;
        TPWrite "Til_felt=" \Num:=Til_felt;
        Opptatt;
    ENDPROC

    ! Denne sjekker om ruten på brettet har en brikke på seg eller ikke.
    PROC Opptatt()
        CONST num th:=20; ! avstandet fra senter av feltet

        ! Setter at ingen brikker står på brettet
             FOR i FROM 1 TO 64 DO
                 TargetA{i}.opptatt := false;
             ENDFOR

             ! Sjekker en brikke av gangen om gangen om den står på et av de 64 feltene
             ! Hvis brikka står på et av feltene bil TargetA{j}.opptatt := TRUE
                  FOR i FROM 1 TO 32 DO
                      FOR j FROM 1 TO 64 DO
                            IF TargetA{j}.target.trans.x-th < brikke{i}.trans.x  AND  TargetA{j}.target.trans.x + th > brikke{i}.trans.x AND TargetA{j}.target.trans.y-th < brikke{i}.trans.y  AND  TargetA{j}.target.trans.y + th > brikke{i}.trans.y THEN
                                TargetA{j}.opptatt := TRUE;
                            ENDIF
                      ENDFOR
                  ENDFOR
         ENDPROC



    ! prosessen for å spille, denne henter opp andre prosesser som den trenger.
    PROC spille ()

        VAR num th:=20; ! Hvor stor toleranse vi godtar for plasering til brikken

        ! Sjekker hvilke felt som er opptatt
        Opptatt;

        ! Hvis feltet er opptatt, skal brikken som står på plassen slås ut
        IF TargetA{Til_felt}.opptatt THEN
            ! finner hvilken brikke som står på plassen med denne for-løkken og if-statment om brikken har posisjon i innenfor 5mm av feltet.
            FOR i FROM 1 TO 32 DO
                IF (TargetA{Til_felt}.target.trans.x-th < brikke{i}.trans.x  AND  TargetA{Til_felt}.target.trans.x + th > brikke{i}.trans.x AND TargetA{Til_felt}.target.trans.y-th < brikke{i}.trans.y  AND  TargetA{Til_felt}.target.trans.y + th > brikke{i}.trans.y) THEN
                    brikke_ut:=i;
                ENDIF
            ENDFOR
                ! Funnet riktig brikke og slår ut den
                Sla_ut;
                ! flytter brikken til den nye ledige plassen.
            move;

        ! Hvis plassen er ledig flytter brikke til den nye plassen
        ELSE
            move;
        ENDIF

    ENDPROC

    ! Denne prosessen flytter brikker som blir slått ut til en lagringsplass på siden av brettet
    PROC Sla_ut ()
        CONST num lager_x:= 55;
        CONST num lager_y:= 100;
        IF lager1>6 THEN ! Denne IF lager en ny kolonne når det er slått ut flere enn 7 brikker
            lager2:=lager2+1;
            lager1:=0;
        ENDIF

        ! Henter brikke som blir slått ut
        MoveJ Offs(brikke{brikke_ut},0,0,-100-brikke{brikke_ut}.trans.z),Speed_hor,fine,picker\WObj:=board2;
        MoveL brikke{brikke_ut},Speed_ned,fine,picker\WObj:=board2;
        Set DO10_1;
        WaitTime(tid);
        MoveL Offs(brikke{brikke_ut},0,0,-100-brikke{brikke_ut}.trans.z),Speed_opp,fine,picker\WObj:=board2;

        ! Flytter brikke til lagringsplass på siden av brettet
        MoveL Offs(TargetA{1}.target,lager_x*lager1,lager_y*lager2,-100),Speed_hor,fine,picker\WObj:=board2;
        MoveL Offs(TargetA{1}.target,lager_x*lager1,lager_y*lager2,brikke{brikke_ut}.trans.z),Speed_ned,fine,picker\WObj:=board2;
        reset DO10_1;
        WaitTime(tid);
        MoveL Offs(TargetA{1}.target,lager_x*lager1,lager_y*lager2,-100),Speed_opp,fine,picker\WObj:=board2;

        ! Lagrer informasjon om hvor brikken som er slått ut står nå
        brikke{brikke_ut}:=OFFS(TargetA{1}.target,lager_x*lager1,lager_y*lager2,brikke{brikke_ut}.trans.z);
        lager1:=lager1+1;
        Opptatt;
        ! Skriver ut hvilken brikke som er flyttet
        TPWrite "brikke " \Num:=brikke_flytt;
    ENDPROC

    ! Denne prosessen brukes for sette roboten i en trygg poseisjon.
    ! Venter på at en av knappen ved roboten blir trykket for å fortsette/komme ut av while loopen.
    PROC while_hold()
        safe_pose;
        HOLD:=0;
        WHILE HOLD = 0 DO
            set DO10_8;
        ENDWHILE
        Reset DO10_8;
    ENDPROC

    ! Denne prosessen brukes for å sende roboten til en trygg posisjon slik at vi kan ta bilder.
    PROC safe_pose()
        MoveJ [[0,0,0],[1,0,0,0],[0,0,2,0],[9E+09,9E+09,9E+09,9E+09,9E+09,9E+09]],v500,fine,picker\WObj:=safepose;
    ENDPROC

ENDMODULE

--- Backups/IRB140_6_81/SYSPAR/EIO.cfg ---
EIO:CFG_1.0:6:1::
#
EIO_SIGNAL:

      -Name "DO10_1" -SignalType "DO"

      -Name "DO10_8" -SignalType "DO"

      -Name "DI10_15" -SignalType "DI"

      -Name "DI10_16" -SignalType "DI"

      -Name "DI10_1" -SignalType "DI"

      -Name "DI10_2" -SignalType "DI"
